TYPE ST_ProcessDoor_CMD :
STRUCT
	
	Extend				: BOOL;		
	Retract				: BOOL;		
	
END_STRUCT
END_TYPE

(* stored: Version 1.1.0.1, ProductVersion 3.1.4024.13
   DUT ST_ProcessDoor_CMD: Id {4d3e5f95-7477-4aaa-ade9-ea6a5dd1bafd} *)
